FUNCTION_BLOCK Pizza
VAR
	Exists :BOOL;
	IsBacked:BOOL;
	BakingTime:Time;
END_VAR

END_FUNCTION_BLOCK

(* stored: Version 1.1.0.1, ProductVersion 3.1.4024.3
   POU Pizza: Id {2f80c2d8-2e09-43ca-bf13-fda285a0af48}, SpecialFunc None *)
